TYPE UDT_VacuumInput :
STRUCT
	ActiveIN: BOOL; 
	ActiveOut: BOOL;
	Sensor: BOOL;
	CheckTime: DINT;
	BlowTime: DINT;
	HmiIN: BOOL;
	HmiOut: BOOL;
	Reset: BOOL;
END_STRUCT
END_TYPE

(* stored: Version 1.1.0.1, ProductVersion 3.1.4022.16
   DUT UDT_VacuumInput: Id {e31f8e82-3e1b-4fd3-af90-abb59a082c26} *)
